// TIA Portal V19 export
DATA_BLOCK "A03_DEBUG"   // DB165
// stored: MemoryReserve 100
   VAR
      Force_Sinamics_Infeed_ON : Bool;
      Force_Sinamics_Drives_CtrlSafe : Bool;
      Forse_Contactors_CtrlSafe : Bool;
      LsStratoDepositato : Bool;
      CIn_Manager_DEBUG : Struct
         PareggiatoreTesta : Struct
            Ax : "Positioning_EPOS_Machine_COut";
         END_STRUCT;
         PareggiatoreCoda : Struct
            Ax : "Positioning_EPOS_Machine_COut";
         END_STRUCT;
         Spalle : Struct
            Testa : Struct
               Ax : "Positioning_DOL_Machine_COut";
            END_STRUCT;
            Coda : Struct
               Ax : "Positioning_DOL_Machine_COut";
            END_STRUCT;
         END_STRUCT;
         Spintore : Struct
            Vrt : "ValveMachine_COut";
            Orz : "ValveMachine_COut";
         END_STRUCT;
         TraslazioneStrato : Struct
            Ax_Testa : "Positioning_EPOS_Machine_COut";
            Ax_Coda : "Positioning_EPOS_Machine_COut";
            Manip_Sostegno : "ValveMachine_COut";
            Manip_Pareggiatore : "ValveMachine_COut";
            SostegnoVrt : "ValveMachine_COut";
         END_STRUCT;
         Sollevamento : Struct
            Ax_Testa : "Positioning_DOL_Machine_COut";
            Ax_Coda : "Positioning_DOL_Machine_COut";
         END_STRUCT;
         Sostegno : Struct
            Testa : Struct
               Ax : "Positioning_DOL_Machine_COut";
               Paletto : Struct
                  CtrlSafe : Bool;
                  Standstill : Bool;
                  Rest_CheckNext : Bool;
                  Work_CheckNext : Bool;
                  Pos : Int;
                  RestPosition : Bool;
               END_STRUCT;
            END_STRUCT;
            Coda : Struct
               Ax : "Positioning_DOL_Machine_COut";
               Paletto : Struct
                  CtrlSafe : Bool;
                  Standstill : Bool;
                  Rest_CheckNext : Bool;
                  Work_CheckNext : Bool;
                  Pos : Int;
                  RestPosition : Bool;
               END_STRUCT;
            END_STRUCT;
         END_STRUCT;
         Navetta : Struct
            ReadyToRecive : Bool;
            OutOfWorkspace : Bool;
            InPosizioneDiDeposito : Bool;
            RequestDeposito : Bool;
         END_STRUCT;
         RegolazBord : Struct
            CassettaOP : Real := 65.0;
            LineSetupExe : Bool;
         END_STRUCT;
      END_STRUCT;
      CIn_Manager04_Debug : Struct
         Navetta : Struct
            Testa : Struct
               Ax : "Positioning_DOL_Machine_COut";
               PalettiEsterni : "ValveMachine_COut";
               PalettiInterni : "ValveMachine_COut";
            END_STRUCT;
            Coda : Struct
               Ax : "Positioning_DOL_Machine_COut";
               PalettiEsterni : "ValveMachine_COut";
               PalettiInterni : "ValveMachine_COut";
            END_STRUCT;
            Cumulativo : Struct
               PalettiEsterni : "ValveMachine_COut";
               PalettiInterni : "ValveMachine_COut";
            END_STRUCT;
         END_STRUCT;
         Sollevamento : Struct
            ReadyToDrop : Bool;   // In posizione di deposito e pacco completato
         END_STRUCT;
         Antiribaltamento : Struct
            Work : Bool;
            Rest : Bool;
         END_STRUCT;
      END_STRUCT;
   END_VAR
   VAR RETAIN
      HU_Test : Struct
         Enable : Bool;
         EnableDrive : Bool;
         "Req_Par-Bloccaggio" : Bool;
         "Req_Par-Paregg" : Bool;
         Ctrl_Safe : Bool;
      END_STRUCT;
   END_VAR
   VAR
      test_bitA : Bool;
      test_bitB : Bool;
   END_VAR
   VAR RETAIN
      A0301_Manager : Struct
         BeamCode : Bool;   // 0=Solo Part / 1 = Accoppiamento Part
         "Case" : Int;
         "P1-P3_Init" : Bool;
         "P1-P2_Init" : Bool;
         TrasportoStart : Bool;
         PTrk_Pos1_Write : Bool;
      END_STRUCT;
      A0302_Manager : Struct
         BeamCode : Bool;   // 0=Solo Part / 1 = Accoppiamento Part
         JMP : Bool := TRUE;
         A0303_ReadyToRecive : Bool;
         PareggiaRead : Bool;
         AttrezzamentoBordatrice : Bool;
         BTrk_EXIT_Clear : Bool;
      END_STRUCT;
   END_VAR
   VAR
      A301_PTrk : "PTrk_Item";
   END_VAR
BEGIN
   A301_PTrk.O_ID := 1;
   A301_PTrk.C_ID := 0;
   A301_PTrk.Quality := 0;
   A301_PTrk.Beam_Code := 1;
   A301_PTrk.PLen_Meas := 2700.0;
   A301_PTrk.W_A := 140.0;
   A301_PTrk.H_B := 4.5;
   A301_PTrk.ShiftDone := FALSE;
END_DATA_BLOCK
